_CFC_ (* Continuous Function Chart, elements in execution order *)
#0 TON_YA1_AVT:TON(IN: SHU6_PV1_1YA1_DI5_A, PT: T#10s)
#1 AND(SHU6_PV1_MV1_DI2_RUN, SHU6_PV1_YA1_DI3_ZKR)
#2 INT_TO_TIME(ZADER_SHU6_PV1_YA1_DI4_OTK)
#3 MUL(#2, 1000)
#4 TON_YA1_OTKR:TON(IN: #1, PT: #3)
#5 AND(NOT SHU6_PV1_MV1_DI2_RUN, SHU6_PV1_YA1_DI4_OTK)
#6 INT_TO_TIME(ZADER_SHU6_PV1_YA1_DI3_ZKR)
#7 MUL(#6, 1000)
#8 TON_YA1_ZKR:TON(IN: #5, PT: #7)
#9 AND(SHU6_PV1_MV1_DI2_RUN, NOT SHU6_PV1_YA1_DI4_OTK)
#10 INT_TO_TIME(ZADER_SHU6_PV1_YA1_DI4_OTK)
#11 MUL(#10, 1000)
#12 TON_YA1_NE_OTKR:TON(IN: #9, PT: #11)
#13 AND(NOT SHU6_PV1_MV1_DI2_RUN, NOT SHU6_PV1_YA1_DI3_ZKR)
#14 INT_TO_TIME(ZADER_SHU6_PV1_YA1_DI3_ZKR)
#15 MUL(#14, 1000)
#16 TON_YA1_NE_ZAKR:TON(IN: #13, PT: #15)
#17 OR(#4.Q, #8.Q, #12.Q, #16.Q, YA1_OTKAZ)
#18 AND(#0.Q, #17)
#19 SR_YA1_OTKAZ:SR(SET1: #18, RESET: SHU6_PV1_SB)
#20 SHU6_PV1_Z_YA1_OTKAZ <= #19.Q1
_END_CFC_
(* the same logic as Structured Text *)
TON_YA1_AVT(IN := SHU6_PV1_1YA1_DI5_A, PT := T#10s);
TON_YA1_OTKR(IN := SHU6_PV1_MV1_DI2_RUN AND SHU6_PV1_YA1_DI3_ZKR, PT := INT_TO_TIME(ZADER_SHU6_PV1_YA1_DI4_OTK) * 1000);
TON_YA1_ZKR(IN := NOT SHU6_PV1_MV1_DI2_RUN AND SHU6_PV1_YA1_DI4_OTK, PT := INT_TO_TIME(ZADER_SHU6_PV1_YA1_DI3_ZKR) * 1000);
TON_YA1_NE_OTKR(IN := SHU6_PV1_MV1_DI2_RUN AND NOT SHU6_PV1_YA1_DI4_OTK, PT := INT_TO_TIME(ZADER_SHU6_PV1_YA1_DI4_OTK) * 1000);
TON_YA1_NE_ZAKR(IN := NOT SHU6_PV1_MV1_DI2_RUN AND NOT SHU6_PV1_YA1_DI3_ZKR, PT := INT_TO_TIME(ZADER_SHU6_PV1_YA1_DI3_ZKR) * 1000);
SR_YA1_OTKAZ(SET1 := TON_YA1_AVT.Q AND (TON_YA1_OTKR.Q OR TON_YA1_ZKR.Q OR TON_YA1_NE_OTKR.Q OR TON_YA1_NE_ZAKR.Q OR YA1_OTKAZ), RESET := SHU6_PV1_SB);
SHU6_PV1_Z_YA1_OTKAZ := SR_YA1_OTKAZ.Q1;
END_PROGRAM

(* POU TZBiS/TZB/Z_YA2_Otk, CFC *)
PROGRAM Z_YA2_Otk
VAR
	SR_YA2_OTKAZ: SR;
	TON_YA2_AVT: TON;
	TON_YA2_OTKR: TON;
	TON_YA2_ZKR: TON;
	TON_YA2_NE_OTKR: TON;
	TON_YA2_NE_ZKR: TON;
END_VAR
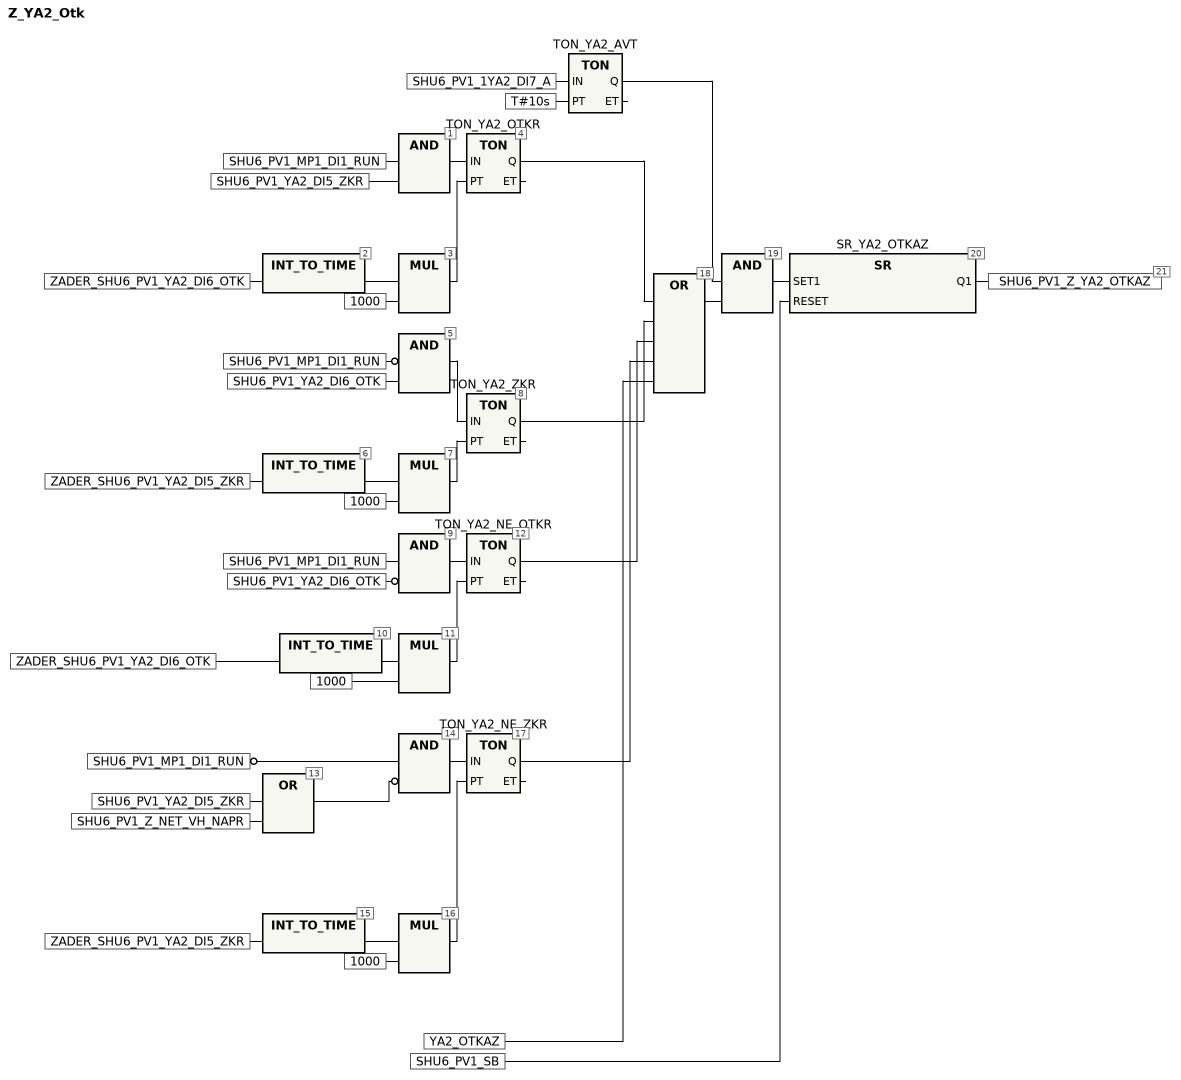
_CFC_ (* Continuous Function Chart, elements in execution order *)
#0 TON_YA2_AVT:TON(IN: SHU6_PV1_1YA2_DI7_A, PT: T#10s)
#1 AND(SHU6_PV1_MP1_DI1_RUN, SHU6_PV1_YA2_DI5_ZKR)
#2 INT_TO_TIME(ZADER_SHU6_PV1_YA2_DI6_OTK)
#3 MUL(#2, 1000)
#4 TON_YA2_OTKR:TON(IN: #1, PT: #3)
#5 AND(NOT SHU6_PV1_MP1_DI1_RUN, SHU6_PV1_YA2_DI6_OTK)
#6 INT_TO_TIME(ZADER_SHU6_PV1_YA2_DI5_ZKR)
#7 MUL(#6, 1000)
#8 TON_YA2_ZKR:TON(IN: #5, PT: #7)
#9 AND(SHU6_PV1_MP1_DI1_RUN, NOT SHU6_PV1_YA2_DI6_OTK)
#10 INT_TO_TIME(ZADER_SHU6_PV1_YA2_DI6_OTK)
#11 MUL(#10, 1000)
#12 TON_YA2_NE_OTKR:TON(IN: #9, PT: #11)
#13 OR(SHU6_PV1_YA2_DI5_ZKR, SHU6_PV1_Z_NET_VH_NAPR)
#14 AND(NOT SHU6_PV1_MP1_DI1_RUN, NOT #13)
#15 INT_TO_TIME(ZADER_SHU6_PV1_YA2_DI5_ZKR)
#16 MUL(#15, 1000)
#17 TON_YA2_NE_ZKR:TON(IN: #14, PT: #16)
#18 OR(#4.Q, #8.Q, #12.Q, #17.Q, YA2_OTKAZ)
#19 AND(#0.Q, #18)
#20 SR_YA2_OTKAZ:SR(SET1: #19, RESET: SHU6_PV1_SB)
#21 SHU6_PV1_Z_YA2_OTKAZ <= #20.Q1
_END_CFC_
(* the same logic as Structured Text *)
TON_YA2_AVT(IN := SHU6_PV1_1YA2_DI7_A, PT := T#10s);
TON_YA2_OTKR(IN := SHU6_PV1_MP1_DI1_RUN AND SHU6_PV1_YA2_DI5_ZKR, PT := INT_TO_TIME(ZADER_SHU6_PV1_YA2_DI6_OTK) * 1000);
TON_YA2_ZKR(IN := NOT SHU6_PV1_MP1_DI1_RUN AND SHU6_PV1_YA2_DI6_OTK, PT := INT_TO_TIME(ZADER_SHU6_PV1_YA2_DI5_ZKR) * 1000);
TON_YA2_NE_OTKR(IN := SHU6_PV1_MP1_DI1_RUN AND NOT SHU6_PV1_YA2_DI6_OTK, PT := INT_TO_TIME(ZADER_SHU6_PV1_YA2_DI6_OTK) * 1000);
TON_YA2_NE_ZKR(IN := NOT SHU6_PV1_MP1_DI1_RUN AND NOT (SHU6_PV1_YA2_DI5_ZKR OR SHU6_PV1_Z_NET_VH_NAPR), PT := INT_TO_TIME(ZADER_SHU6_PV1_YA2_DI5_ZKR) * 1000);
SR_YA2_OTKAZ(SET1 := TON_YA2_AVT.Q AND (TON_YA2_OTKR.Q OR TON_YA2_ZKR.Q OR TON_YA2_NE_OTKR.Q OR TON_YA2_NE_ZKR.Q OR YA2_OTKAZ), RESET := SHU6_PV1_SB);
SHU6_PV1_Z_YA2_OTKAZ := SR_YA2_OTKAZ.Q1;
END_PROGRAM

(* POU TZBiS/TZB/Z_YA3_Otk, CFC *)
PROGRAM Z_YA3_Otk
VAR
	SR_YA2_Otk: SR;
	TON_YA3_Rassog: TON;
	RT_Rassog: R_TRIG;
	TON_YA3_Rassog1: TON;
	TIME_DELAY: TIME;
END_VAR
VAR (* helpers for the ST form of the networks *)
	_t14 : BOOL;
	_t84 : BOOL;
	_t140 : BOOL;
END_VAR
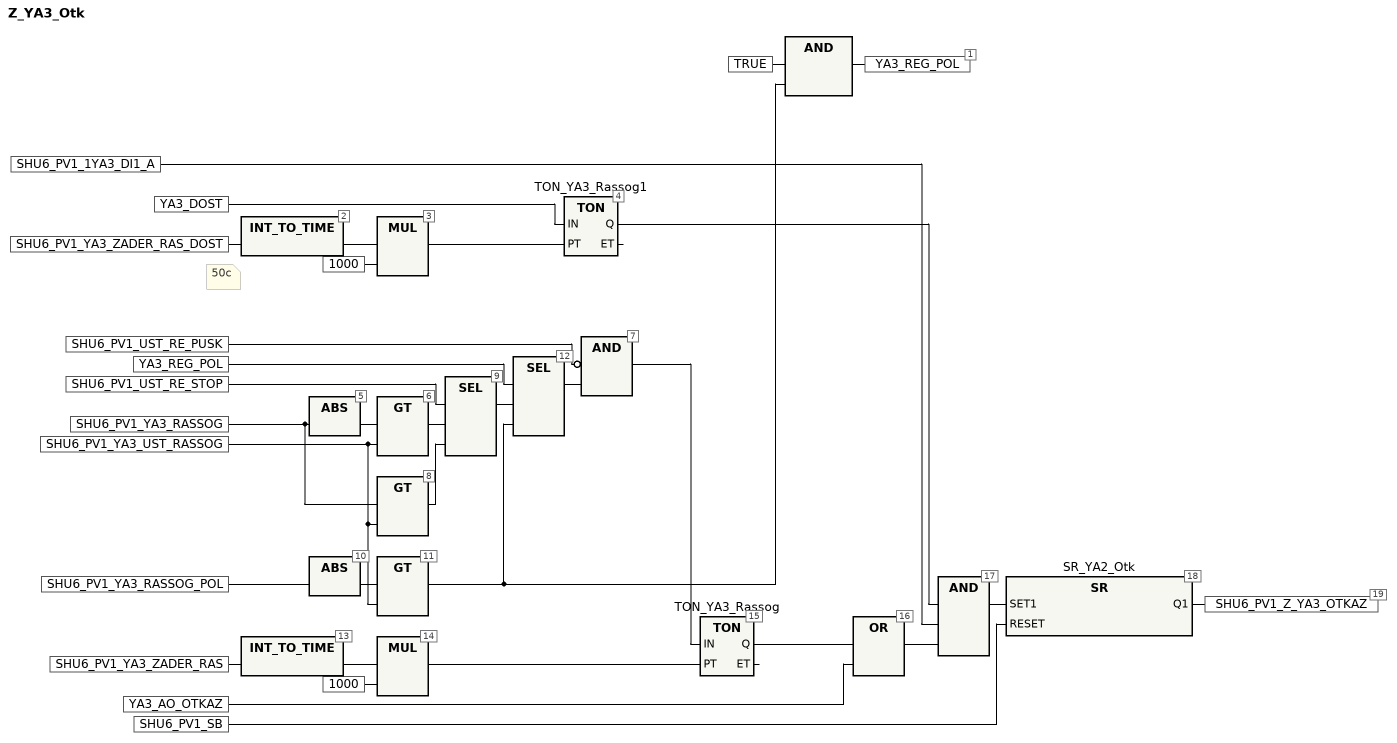
